SUBAPPLICATION AuxIXA_TO_logiBUS_QXA_BG (* AUX-Funktion (Aux_IXA) auf DigitalOutput QXA mit GreenWhiteBackground. Generisch, analog zu Button_IXA_TO_logiBUS_QXA_BG (dort Button statt AUX). *)
  (* Standard: 61499-2 *)
  (* Version 1.0, 2026-09-09, Franz Höpfinger, Meisterschulen am Ostbahnhof, Ausgelagert aus Uebung_010f2_sub_AX zur Wiederverwendung. *)
  PACKAGE MyLib::sys;
  IMPORT isobus::UT::Q::const::IDs::ID_NULL;
  IMPORT logiBUS::io::DQ::logiBUS_DO;
  IMPORT logiBUS::io::DQ::logiBUS_DO_S;
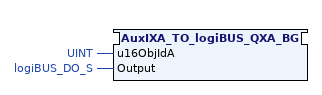
  VAR_INPUT
    u16ObjIdA : UINT := ID_NULL; (* Object ID AUX *)
    Output : logiBUS::io::DQ::logiBUS_DO_S := logiBUS_DO::Invalid; (* Identify the Output Output_Q1..Q8 *)
  END_VAR
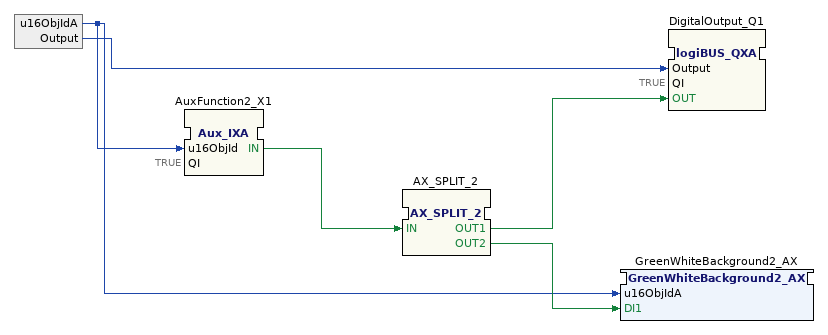
  FBS
    DigitalOutput_Q1 : logiBUS::io::DQ::logiBUS_QXA(QI := TRUE);
    AuxFunction2_X1 : isobus::UT::io::Auxiliary::IN::Aux_IXA(QI := TRUE);
    AX_SPLIT_2 : adapter::events::unidirectional::AX_SPLIT_2;
  END_FBS
  SUBAPPS
    GreenWhiteBackground2_AX : MyLib::sys::GreenWhiteBackground2_AX;
  END_SUBAPPS
  DATA_CONNECTIONS
    u16ObjIdA TO AuxFunction2_X1.u16ObjId;
    u16ObjIdA TO GreenWhiteBackground2_AX.u16ObjIdA;
    Output TO DigitalOutput_Q1.Output;
  END_CONNECTIONS
  ADAPTER_CONNECTIONS
    AuxFunction2_X1.IN TO AX_SPLIT_2.IN;
    AX_SPLIT_2.OUT1 TO DigitalOutput_Q1.OUT;
    AX_SPLIT_2.OUT2 TO GreenWhiteBackground2_AX.DI1;
  END_CONNECTIONS
END_SUBAPPLICATION
